FUNCTION "LGF_MergeBitsToByte" : Byte
TITLE = LGF_MergeBitsToByte
{ S7_Optimized_Access := 'TRUE' }
AUTHOR : Siemens_Digital_Industry
FAMILY : LGF
NAME : LGF_MergeBitsToByte
//This function merge 8 Bits / 8 Boolean variables into one Byte variable.
   VAR_INPUT
      bit7 : Bool;   // Input Bit 7 - MSB
      bit6 : Bool;   // Input Bit 6
      bit5 : Bool;   // Input Bit 5
      bit4 : Bool;   // Input Bit 4
      bit3 : Bool;   // Input Bit 3
      bit2 : Bool;   // Input Bit 2
      bit1 : Bool;   // Input Bit 1
      bit0 : Bool;   // Input Bit 0 - LSB
   END_VAR

   VAR_TEMP
      tempByte : Byte;   // Temp memory to merge Bits into a Byte
   END_VAR


BEGIN
	REGION BLOCK INFO HEADER
	  //===============================================================================
	  // SIEMENS AG / (c)Copyright 2018
	  //-------------------------------------------------------------------------------
	  // Title:            LGF_MergeBitsToByte
	  // Comment/Function: This function merge 8 Bits / 8 Boolean variables into one Byte variable.
	  // Library/Family:   LGF (Library General Functions)
	  // Author:           Siemens Digital Industry Support
	  // Tested with:      S7-PLCSIM Advanced V2.0 SP1
	  // Engineering:      TIA Portal V14 / V14SP1
	  // Restrictions:     ENO disabled - no error handling, no failure possible.
	  // Requirements:     PLC (S7-1200 / S7-1500)
	  //-------------------------------------------------------------------------------
	  // Change log table:
	  // Version  | Date       | Expert in charge       | Changes applied
	  //----------|------------|------------------------|------------------------------
	  // 01.00.00 | 20.06.2019 | Simatic Systems Support
	  //                         First release
	  // 03.00.00 | 23.04.2020 | Simatic Systems Support | Set version to V3.0.0
	  //                         harmonize the version of the whole library
	  // 03.00.01 | 22.02.2021 | Simatic Systems Support
	  //                         Insert documentation
	  //=============================================================================
	END_REGION

	REGION MERGE
	  // set the bits by slice access
	  #tempByte.%X7 := #bit7;
	  #tempByte.%X6 := #bit6;
	  #tempByte.%X5 := #bit5;
	  #tempByte.%X4 := #bit4;
	  #tempByte.%X3 := #bit3;
	  #tempByte.%X2 := #bit2;
	  #tempByte.%X1 := #bit1;
	  #tempByte.%X0 := #bit0;
	END_REGION

	REGION OUTPUT
	  #LGF_MergeBitsToByte := #tempByte;
	  // no error handling needed
	  ENO := TRUE;
	END_REGION

END_FUNCTION

